(* IEC 61131-3 sources: InfiniteStateMachine/st/infinitestatemachine/function_blocks/statemachine, 3 files *)

(* ---- in-In.st ---- *)
(* --- Interface --- *)
METHOD In : BOOL
VAR_INPUT
	itfState: IState;
END_VAR
VAR
	iLevel : INT := 0;
END_VAR
(* --- Implementation --- *)
(*
 * The following do-while loop's condition assumes early-out semantics.
 * It assumes that the second sub-condition does *not* evaluate unless the first sub-condition is true.
 *)
WHILE iLevel < iDepth AND itfStates[iLevel] <> itfState DO
	iLevel := iLevel + 1;
END_WHILE
In := iLevel < iDepth;

(* ---- leave-Leave.st ---- *)
(* --- Interface --- *)
METHOD PROTECTED Leave
VAR_INPUT
END_VAR
VAR
	itfState : IState;
END_VAR

(* --- Implementation --- *)
itfState := Pop();
IF itfState <> 0 THEN
	itfState.Leave(THIS^);
END_IF

(* ---- push-Push.st ---- *)
(* --- Interface --- *)
METHOD PROTECTED Push : BOOL
VAR_INPUT
	itfState : IState;
END_VAR

(* --- Implementation --- *)
Push := iDepth < ISM.gc_iMaxDepth;
IF Push THEN
	itfStates[iDepth] := itfState;
	iDepth := iDepth + 1;
END_IF
